INTERFACE ITF_TcpIpBase

METHOD ConnectToRobot : BOOL
VAR_INPUT
END_VAR
END_METHOD

METHOD DisconnectFromRobot : BOOL
VAR_INPUT
END_VAR
END_METHOD

METHOD GetData : ARRAY[0..1439] OF byte
VAR_INPUT
END_VAR
END_METHOD

METHOD IsConnected : BOOL
VAR_INPUT
END_VAR
END_METHOD

PROPERTY RemoteServerIP : T_IPv4Addr
GET
END_GET
SET
END_SET
END_PROPERTY

PROPERTY RemoteServerPort : UDINT
GET
END_GET
SET
END_SET
END_PROPERTY

END_INTERFACE

(* stored: Version 1.1.0.1, ProductVersion 3.1.4024.12
   Itf ITF_TcpIpBase: Id {dfd1e5fa-86c5-4f58-ab3f-80e1a76b8c9d}
   Method ConnectToRobot: Id {35ea5ab8-974d-42a5-b03e-607e992f079b}
   Method DisconnectFromRobot: Id {662981ab-d0c1-4edb-a455-182e81a4a8a0}
   Method GetData: Id {a886064e-36c9-4552-b51b-d151470a81bb}
   Method IsConnected: Id {ff1b670a-ddaf-46b6-876f-7ff81f11c828}
   Property RemoteServerIP: Id {9d868d5b-2200-4ec8-b3f7-7549f74a96e1}
   Get Get: Id {fd822b0b-03e4-4319-ba90-1eaf45fdf61c}
   Set Set: Id {85870ea8-aeea-48eb-94cb-48378570f79e}
   Property RemoteServerPort: Id {19cf41cb-9661-4dec-ad1d-9bdc18b9c542}
   Get Get: Id {d0774186-68c0-432d-a4a9-caffbebe2cca}
   Set Set: Id {dd16c6bb-0cf5-4588-b586-68f75f14a87a} *)
